(* IEC 61131-3 sources: AutomationStudio/SuszarkaDoRak, 3 files *)

(* ---- Types.typ ---- *)
TYPE
	BathRoomTyp: STRUCT
		Suszarka : DryerTyp;
	END_STRUCT;

	DryerTyp: STRUCT
		diHand : BOOL; (* Sensor wykrywajacy onbecnosc rak *)
		doDmuchawa: BOOL; (* Wysterowanie cewki stycznika -> grzałka + wentylator 220vac *)
		diTermik : BOOL; (* Termostat wykrywający za gorące styki stycznika *)
	END_STRUCT;

	BathRoomParTyp: STRUCT
		Suszarka : DryerParTyp;
	END_STRUCT;

	DryerParTyp: STRUCT
		uiCzasON : REAL; (*Deklaracja czasu załączenie sek ->GUI *)
		uiCzasOFF: REAL; (*Deklaracja przerw sek ->GUI *)
		uiCzasPracy: WorkTimeTyp; (*Łączny czas pracy szuszarki w trybie suszenia h,m*)
		uiLiczbaOnOff : DINT; (* Liczba załączeń suszarki *)
	END_STRUCT;

	WorkTimeTyp: STRUCT
		uiGodziny: REAL;
		uiSekundy: REAL;
		uiMinuty: REAL;
	END_STRUCT;

END_TYPE

(* ---- Main.st ---- *)
PROGRAM _INIT
	(* Insert code here *)

END_PROGRAM

PROGRAM _CYCLIC
	(* Insert code here *)

	ZegarTOF[0].IN:=Lazienka[0].Suszarka.diHand;
	ZegarTOF[0].PT:=REAL_TO_TIME(LazienkaPar[0].Suszarka.uiCzasOFF*1000); //GUI -> sekundy ->TIME
	ZegarTOF[0]();

	ZegarTON[0].IN:=ZegarTOF[0].Q;;
	ZegarTON[0].PT:=REAL_TO_TIME(LazienkaPar[0].Suszarka.uiCzasON*1000); //GUI -> sekundy ->TIME
	ZegarTON[0](); //Function update Block -> exe
	Lazienka[0].Suszarka.doDmuchawa:=ZegarTON[0].Q AND ZegarTOF[0].Q AND NOT(Lazienka[0].Suszarka.diTermik);

	IF EDGEPOS(Lazienka[0].Suszarka.doDmuchawa) THEN (*edgepos zbocza narastające*);
		LazienkaPar[0].Suszarka.uiLiczbaOnOff:=LazienkaPar[0].Suszarka.uiLiczbaOnOff+1;
	END_IF

	ZegarTON[1].IN:=NOT(ZegarTON[1].Q) AND Lazienka[0].Suszarka.doDmuchawa ;
	ZegarTON[1].PT:=T#1s;
	ZegarTON[1](); //generator sekund pierwszy sposób odlicznczania

	IF ZegarTON[1].Q THEN
		LazienkaPar[0].Suszarka.uiCzasPracy.uiSekundy:=LazienkaPar[0].Suszarka.uiCzasPracy.uiSekundy+1;
	END_IF

	IF LazienkaPar[0].Suszarka.uiCzasPracy.uiSekundy>=60 THEN
		LazienkaPar[0].Suszarka.uiCzasPracy.uiMinuty:=LazienkaPar[0].Suszarka.uiCzasPracy.uiMinuty+1;
		LazienkaPar[0].Suszarka.uiCzasPracy.uiSekundy:=0;
	END_IF

	IF LazienkaPar[0].Suszarka.uiCzasPracy.uiMinuty>=60 THEN
		LazienkaPar[0].Suszarka.uiCzasPracy.uiGodziny:=LazienkaPar[0].Suszarka.uiCzasPracy.uiGodziny+1;
		LazienkaPar[0].Suszarka.uiCzasPracy.uiMinuty:=0;
	END_IF

	IF (((TIME_TO_DINT(ZegarTON[0].ET) MOD 1000)=0) AND (TIME_TO_DINT(ZegarTON[0].ET)>0) AND (Lazienka[0].Suszarka.doDmuchawa)) THEN
		LazienkaPar[1].Suszarka.uiCzasPracy.uiSekundy:=LazienkaPar[1].Suszarka.uiCzasPracy.uiSekundy+1;
	END_IF

	IF LazienkaPar[1].Suszarka.uiCzasPracy.uiSekundy>=60 THEN
		LazienkaPar[1].Suszarka.uiCzasPracy.uiMinuty:=LazienkaPar[1].Suszarka.uiCzasPracy.uiMinuty+1;
		LazienkaPar[1].Suszarka.uiCzasPracy.uiSekundy:=0;
	END_IF

	IF LazienkaPar[1].Suszarka.uiCzasPracy.uiMinuty>=60 THEN
		LazienkaPar[1].Suszarka.uiCzasPracy.uiGodziny:=LazienkaPar[1].Suszarka.uiCzasPracy.uiGodziny+1;
		LazienkaPar[1].Suszarka.uiCzasPracy.uiMinuty:=0;
	END_IF

END_PROGRAM

PROGRAM _EXIT
	(* Insert code here *)

END_PROGRAM

(* ---- Variables.var ---- *)
VAR
	Lazienka : ARRAY[0..1] OF BathRoomTyp;
	ZegarTON : ARRAY[0..9] OF TON; (*Deklaracja funkcji zegara TON*)
	ZegarTOF : ARRAY[0..9] OF TOF; (*Deklaracja funkcji zegara TOF*)(*on się uzbraja jak dajemy 1 i jak damy zaero to odlicza*)

END_VAR

VAR RETAIN
	LazienkaPar : ARRAY[0..1] OF BathRoomParTyp;
END_VAR
